TYPE DS_EventHistoryLogToFile EXTENDS DS_EventHistory :
STRUCT
	sEventCode						: STRING(10);
	sEventType						: STRING(10);
	sLocation						: STRING(20);
	sSubLocation					: STRING(20);
	sDescription 					: STRING(80);
END_STRUCT
END_TYPE

(* stored: Version 1.1.0.1, ProductVersion 3.1.4024.12
   DUT DS_EventHistoryLogToFile: Id {ac1753fd-5512-45f8-94b9-c236875cff01} *)
